// SIMATIC S7-200 project (STEP 7-Micro/WIN), CPU 224 REL 01.12

ORGANIZATION_BLOCK 主程序:OB1
TITLE=项目详解
// 系统通过启动按钮启动运行，首先打开进料阀门让棉条进入处理槽，进料过程中由液位传感器实时监控液位，确保液位不超过预设值以防止溢出。进料启用标志只有在液位传感器未检测到满液位且液位未满标志未置位时才会置位。进料完成后，搅拌电机在进料阀门关闭且温度适宜时启动，进行棉条的均匀分布，搅拌时间由搅拌延时定时器精确控制。细纱机运行状态在系统启动后保持置位，直到急停或故障发生。
// 在拉伸纺纱阶段，罗拉电机启动负责拉伸棉条。罗拉电机启动或罗拉电机停止前，纱架升起必须已经置位，以确保棉条正确引导至罗拉，避免纱线断裂。纱架升起在温度传感器1和定时器条件下置位，纱架降下在温度传感器2和定时器条件下置位。若特定标志位置位且定时器未超时，冷却器激活；加热器在进料阀门关闭且温度适宜时启动。出料阀门在标志位复位后开启，以输出纺好的细纱。
BEGIN
Network 1 // 网络标题
// 网络注释
LD     I0.4
O      Q0.0
=      M30.0
?000
Network 2
LD     SM0.1
MOVW   +5001, VW4000
Network 3
LD     M30.0
AN     T102
A      I0.3
=      Q0.0
Network 4
LD     M30.0
LD     I0.4
O      Q0.1
ALD
A      I1.1
AN     Q0.2
A      I0.3
=      Q0.1
Network 5
LD     M30.0
AN     I1.1
AN     M0.0
=      M30.1
Network 6
LD     M30.1
LD     I0.5
O      Q1.0
ALD
=      M30.2
Network 7
LD     M30.2
AN     Q1.1
AN     C1
AN     I0.6
=      Q1.0
Network 8
LD     M30.1
LD     I0.6
O      C1
O      Q1.1
ALD
AN     Q1.0
=      Q1.1
Network 9
LD     Q0.0
LD     I0.7
O      M0.2
ALD
=      M0.2
Network 10
LD     Q0.0
LD     I1.0
O      I1.2
O      M0.2
O      M0.3
O      M6.6
O      M6.7
ALD
=      M0.3
Network 11
LD     Q0.0
LD     I1.5
O      M0.0
ALD
LD     M0.2
O      M0.3
ALD
=      M0.0
Network 12
LD     Q0.0
LD     I1.5
O      M0.0
ALD
LD     M0.2
O      M0.3
ALD
AW=    VW1058, +2
TON    T108, VW1018
TON    T109, VW1020
Network 13
LD     Q0.0
LD     I2.0
AW=    VW1058, +1
LD     T108
AW=    VW1058, +2
OLD
O      Q0.2
ALD
AN     M0.2
AN     Q0.1
A      I1.3
A      M0.3
=      Q0.2
Network 14
LD     Q0.0
LD     I2.1
A      M0.3
AW=    VW1058, +1
LD     T109
A      M0.3
AW=    VW1058, +2
OLD
O      Q0.6
ALD
A      M0.0
=      Q0.6
Network 15
LD     Q0.0
LD     I2.1
A      M0.3
O      Q0.6
ALD
TON    T102, +200
Network 16
LD     Q0.0
A      M0.3
AN     T103
=      Q2.1
Network 17
LD     Q0.0
A      Q1.0
=      Q2.3
Network 18
LD     Q0.0
A      Q1.1
=      Q2.2
Network 19
LD     Q0.0
A      M0.3
AN     T104
TON    T103, +20
Network 20
LD     Q0.0
A      T103
TON    T104, +20
Network 21
LD     Q1.1
O      Q1.0
A      Q0.0
AN     M0.3
=      Q0.3
Network 22
LD     T105
EU
O      M0.5
A      Q0.0
=      M0.5
Network 23
LD     Q0.0
A      I2.2
LD     I2.3
O      Q0.4
O      Q1.1
ALD
AN     M0.3
=      Q0.4
Network 24
LD     M0.3
AN     M0.2
O      I2.5
O      Q0.7
AN     Q0.1
A      I2.6
=      Q0.5
=      Q0.7
Network 25
LD     SM0.1
BMW    VW800, VW1000, 65
R      M10.0, 8
R      M26.0, 1
R      M11.0, 2
MOVD   +0, VD20
MOVW   +0, VW24
Network 26
LD     SM0.1
O      M26.0
MOVD   +0, VD20
MOVW   +0, VW24
MOVB   8, VB20
MOVD   VD1036, VD123
R      M26.0, 1
Network 27
LD     M10.0
AN     M11.0
AN     M11.1
AN     V24.4
MOVD   +0, VD20
MOVW   +0, VW24
MOVB   16#80, VB20
MOVD   VD1040, VD43
R      M10.0, 8
Network 28
LD     M10.1
AN     M11.0
AN     M11.1
AN     V24.4
MOVD   +0, VD20
MOVW   +0, VW24
MOVB   16#40, VB20
MOVD   VD1044, VD63
R      M10.0, 8
Network 29
LD     M10.2
AN     M11.0
AN     M11.1
AN     V24.4
MOVD   +0, VD20
MOVW   +0, VW24
MOVB   16#20, VB20
MOVD   VD1048, VD83
R      M10.0, 8
Network 30
LD     M10.3
AN     M11.0
AN     M11.1
AN     V24.4
MOVD   +0, VD20
MOVW   +0, VW24
MOVB   16#10, VB20
MOVD   VD1052, VD103
R      M10.0, 8
Network 31
LD     M10.4
AN     M11.0
AN     M11.1
AN     V24.4
MOVD   +0, VD20
MOVW   +0, VW24
MOVB   8, VB20
MOVD   VD1036, VD123
R      M10.0, 8
Network 32
LD     M10.5
AN     M11.0
AN     M11.1
AN     V24.4
MOVD   +0, VD20
MOVW   +0, VW24
MOVB   4, VB20
MOVW   VW1000, VW147
R      M10.0, 8
Network 33
LD     V145.2
AW<=   VW147, +4
AW>=   VW147, +1
MOVW   VW147, VW1000
MOVW   VW147, VW800
MOVW   +800, SMW32
MOVB   16#82, SMB31
MOVW   16#1, MW9
MOVW   VW1000, AC0
DECW   AC0
SLW    MW9, AC0
R      V145.2, 1
Network 34
LD     V145.2
LDW>=  VW147, +5
OW=    VW147, +0
ALD
MOVB   8, VB24
R      V145.2, 1
Network 35
LD     M10.6
EU
S      M11.0, 1
Network 36
LDN    V20.0
AB=    VB21, 0
=      M26.2
Network 37
LD     M10.6
AN     M11.1
AN     V24.4
A      M26.2
MOVD   +0, VD20
MOVW   +0, VW24
MOVB   2, VB20
R      M10.0, 8
Network 38
LD     V168.1
MOVW   VW1030, VW182
MOVB   1, VB20
R      V168.1, 1
Network 39
LD     V180.1
MOVW   VW1022, VW202
MOVB   16#80, VB21
R      V180.1, 1
Network 40
LD     V200.1
MOVW   VW1024, VW222
MOVB   16#40, VB21
R      V200.1, 1
Network 41
LD     V220.1
MOVW   VW1026, VW244
MOVB   16#20, VB21
R      V220.1, 1
Network 42
LD     V242.1
MOVW   VW1056, VW263
MOVB   16#10, VB21
R      V242.1, 1
Network 43
LD     V261.1
MOVW   VW1032, VW284
MOVB   8, VB21
R      V261.1, 1
Network 44
LD     V282.1
MOVW   VW1034, VW300
MOVB   4, VB21
R      V282.1, 1
Network 45
LD     V298.1
MOVD   VD5000, VD324
MOVB   2, VB21
R      V298.1, 1
Network 46
LD     V322.1
MOVB   1, VB21
R      V322.1, 1
Network 47
LD     V346.1
S      M26.0, 1
R      M11.0, 1
R      V346.1, 1
R      M10.0, 8
Network 48
LD     I2.4
EU
R      V723.2, 1
R      V402.2, 1
R      V422.2, 1
R      V442.2, 1
R      V462.2, 1
R      V482.2, 1
R      V502.2, 1
R      V522.2, 1
R      V543.2, 1
R      V561.2, 1
R      V580.2, 1
R      V602.2, 1
R      V622.2, 1
R      V642.2, 1
R      V663.2, 1
R      V686.2, 1
R      V703.2, 1
Network 49
LDB>=  VB22, 1
AB<=   VB22, 16#40
OB>=   VB23, 1
OB>=   VB24, 16#10
AN     I2.4
MOVB   4, VB24
Network 50
LDN    I2.4
AN     M11.1
MOVW   +0, VW22
R      V24.4, 4
Network 51
LDN    I2.4
AB=    VB22, 16#80
MOVB   4, VB24
R      V22.7, 1
Network 52
LDN    I2.4
AB=    VB22, 16#40
MOVB   4, VB24
R      V22.6, 1
R      M11.1, 1
Network 53
LD     M10.7
AN     I2.4
MOVD   +0, VD20
MOVW   +0, VW24
MOVB   4, VB24
R      M10.0, 8
Network 54
LD     M10.7
A      I2.4
AN     M11.0
AN     V24.4
MOVD   +0, VD20
MOVW   +0, VW24
MOVB   16#80, VB22
R      M10.0, 8
S      M11.1, 1
Network 55
LD     V368.1
A      I2.4
MOVB   16#40, VB22
R      V368.1, 1
Network 56
LD     V368.1
AN     I2.4
R      V368.1, 1
R      M11.1, 1
R      M10.0, 8
Network 57
LD     V386.2
A      M11.1
A      I2.4
AW<=   VW388, +17
AW>=   VW388, +1
MOVD   +0, VD22
MOVB   16#20, VB22
DECW   VW388
SRD    VD22, VB389
MOVW   +0, VW388
R      V386.2, 1
R      M11.1, 1
R      M10.0, 8
Network 58
LD     V386.2
A      I2.4
LDW>=  VW388, +18
OW=    VW388, +0
ALD
MOVB   8, VB24
MOVW   +0, VW388
R      V386.2, 1
R      M11.1, 1
R      M10.0, 8
Network 59
LD     V386.2
AN     I2.4
R      V386.2, 1
R      M11.1, 1
R      M10.0, 8
Network 60
LDB>=  VB22, 1
AB<=   VB22, 16#20
OB>=   VB23, 1
OB>=   VB24, 16#20
EU
MOVD   VD1040, VD404
MOVD   VD1044, VD424
MOVD   VD1048, VD444
MOVD   VD1052, VD464
MOVD   VD1036, VD484
MOVW   VW1002, VW504
MOVW   VW1004, VW524
MOVW   VW1028, VW545
Network 61
LDB>=  VB22, 1
AB<=   VB22, 16#20
OB>=   VB23, 1
OB>=   VB24, 16#20
EU
MOVD   VD1006, VD563
MOVW   VW1056, VW582
MOVW   VW1014, VW604
MOVW   VW1016, VW624
MOVW   VW1012, VW644
MOVW   VW1010, VW665
MOVW   VW1058, VW688
MOVW   VW1018, VW705
MOVW   VW1020, VW725
Network 62
LD     V402.2
A      I2.4
AD=    VD404, +0
MOVD   VD404, VD1040
MOVD   VD404, VD840
MOVW   +840, SMW32
MOVB   16#83, SMB31
MOVB   16#10, VB22
R      V402.2, 1
Network 63
LD     V402.2
A      I2.4
AD>=   VD404, +1
MOVB   8, VB24
R      V402.2, 1
Network 64
LD     V422.2
A      I2.4
AD=    VD424, +0
MOVD   VD424, VD1044
MOVD   VD424, VD844
MOVW   +844, SMW32
MOVB   16#83, SMB31
MOVB   8, VB22
R      V422.2, 1
Network 65
LD     V422.2
A      I2.4
AD>=   VD424, +1
MOVB   8, VB24
R      V422.2, 1
Network 66
LD     V442.2
A      I2.4
AD=    VD444, +0
MOVD   VD444, VD1048
MOVD   VD444, VD848
MOVW   +848, SMW32
MOVB   16#83, SMB31
MOVB   4, VB22
R      V442.2, 1
Network 67
LD     V442.2
A      I2.4
AD>=   VD444, +1
MOVB   8, VB24
R      V442.2, 1
Network 68
LD     V462.2
A      I2.4
AD=    VD464, +0
MOVD   VD464, VD1052
MOVD   VD464, VD852
MOVW   +852, SMW32
MOVB   16#83, SMB31
MOVB   2, VB22
R      V462.2, 1
Network 69
LD     V462.2
A      I2.4
AD>=   VD464, +1
MOVB   8, VB24
R      V462.2, 1
Network 70
LD     V482.2
A      I2.4
AD=    VD484, +0
MOVD   VD484, VD1036
MOVD   VD484, VD836
MOVW   +836, SMW32
MOVB   16#83, SMB31
MOVB   1, VB22
R      V482.2, 1
Network 71
LD     V482.2
A      I2.4
AD>=   VD484, +1
MOVB   8, VB24
R      V482.2, 1
Network 72
LD     V502.2
A      I2.4
LDW=   VW504, +205
OW=    VW504, +220
OW=    VW504, +240
ALD
MOVW   VW504, VW1002
MOVW   VW504, VW802
MOVW   +802, SMW32
MOVB   16#82, SMB31
MOVB   16#80, VB23
R      V502.2, 1
Network 73
LD     V502.2
A      I2.4
LDW>=  VW504, +206
OW<=   VW504, +219
OW>=   VW504, +221
OW<=   VW504, +239
OW>=   VW504, +241
OW<=   VW504, +204
ALD
MOVB   8, VB24
R      V502.2, 1
Network 74
LD     V522.2
A      I2.4
LDW=   VW524, +200
OW=    VW524, +250
ALD
MOVW   VW524, VW1004
MOVW   VW524, VW804
MOVW   +804, SMW32
MOVB   16#82, SMB31
MOVB   16#40, VB23
R      V522.2, 1
Network 75
LD     V522.2
A      I2.4
LDW>=  VW524, +201
OW<=   VW524, +249
OW>=   VW524, +251
OW<=   VW524, +199
ALD
MOVB   8, VB24
R      V522.2, 1
Network 76
LD     V543.2
A      I2.4
LDW=   VW545, +25
OW=    VW545, +27
ALD
MOVW   VW545, VW1028
MOVW   VW545, VW828
MOVW   +828, SMW32
MOVB   16#82, SMB31
MOVB   16#20, VB23
R      V543.2, 1
Network 77
LD     V543.2
A      I2.4
LDW>=  VW545, +28
OW<=   VW545, +24
ALD
MOVB   8, VB24
R      V543.2, 1
Network 78
LD     V561.2
A      I2.4
AD<=   VD563, +99999
MOVD   VD563, VD1006
MOVD   VD563, VD806
MOVW   +806, SMW32
MOVB   16#83, SMB31
MOVB   16#10, VB23
R      V561.2, 1
Network 79
LD     V561.2
A      I2.4
AD>=   VD563, +100000
MOVB   8, VB24
R      V561.2, 1
Network 80
LD     V580.2
A      I2.4
AW<=   VW582, +999
MOVW   VW582, VW1056
MOVW   VW582, VW856
MOVW   +856, SMW32
MOVB   16#82, SMB31
MOVB   8, VB23
R      V580.2, 1
Network 81
LD     V580.2
A      I2.4
AW>=   VW582, +1000
MOVB   8, VB24
R      V580.2, 1
Network 82
LD     V602.2
A      I2.4
AW<=   VW604, +99
MOVW   VW604, VW1014
MOVW   VW604, VW814
MOVW   +814, SMW32
MOVB   16#82, SMB31
MOVB   4, VB23
R      V602.2, 1
Network 83
LD     V602.2
A      I2.4
AW>=   VW604, +100
MOVB   8, VB24
R      V602.2, 1
Network 84
LD     V622.2
A      I2.4
LDW=   VW624, +1
OW=    VW624, +2
ALD
MOVW   VW624, VW1016
MOVW   VW624, VW816
MOVW   +816, SMW32
MOVB   16#82, SMB31
MOVB   2, VB23
R      V622.2, 1
Network 85
LD     V622.2
A      I2.4
LDW>=  VW624, +3
OW<=   VW624, +0
ALD
MOVB   8, VB24
R      V622.2, 1
Network 86
LD     V642.2
A      I2.4
AW<=   VW644, +600
MOVW   VW644, VW1012
MOVW   VW644, VW812
MOVW   +812, SMW32
MOVB   16#82, SMB31
MOVB   1, VB23
R      V642.2, 1
Network 87
LD     V642.2
A      I2.4
AW>=   VW644, +601
MOVB   8, VB24
R      V642.2, 1
Network 88
LD     V663.2
A      I2.4
AW<=   VW665, +1999
MOVW   VW665, VW1010
MOVW   VW665, VW810
MOVW   +810, SMW32
MOVB   16#82, SMB31
MOVB   16#80, VB24
R      V663.2, 1
Network 89
LD     V663.2
A      I2.4
AW>=   VW665, +2000
MOVB   8, VB24
R      V663.2, 1
Network 90
LD     V686.2
A      I2.4
LDW=   VW688, +2
OW=    VW688, +1
ALD
MOVW   VW688, VW1058
MOVW   VW688, VW858
MOVW   +858, SMW32
MOVB   16#82, SMB31
MOVB   16#40, VB24
R      V686.2, 1
Network 91
LD     V686.2
A      I2.4
LDW>=  VW688, +3
OW=    VW688, +0
ALD
MOVB   8, VB24
R      V686.2, 1
Network 92
LD     V703.2
A      I2.4
AW<=   VW705, +99
MOVW   VW705, VW1018
MOVW   VW705, VW818
MOVW   +818, SMW32
MOVB   16#82, SMB31
MOVB   16#20, VB24
R      V703.2, 1
Network 93
LD     V703.2
A      I2.4
AW>=   VW705, +100
MOVB   8, VB24
R      V703.2, 1
Network 94
LD     V723.2
A      I2.4
AW<=   VW725, +999
MOVW   VW725, VW1020
MOVW   VW725, VW820
MOVW   +820, SMW32
MOVB   16#82, SMB31
MOVB   16#10, VB24
R      V723.2, 1
Network 95
LD     V723.2
A      I2.4
AW>=   VW725, +1000
MOVB   8, VB24
R      V723.2, 1
Network 96
LD     V747.1
A      I2.4
S      M26.0, 1
R      M10.0, 8
R      V747.1, 1
R      V24.4, 1
Network 97
LD     V24.3
O      V24.2
AB=    MB10, 0
TON    T37, +30
Network 98
LD     T37
S      M26.0, 1
Network 99
LD     Q1.0
O      Q1.1
AN     M6.0
TON    T110, +600
Network 100
LD     T110
EU
=      M6.0
Network 101
LD     Q1.0
O      Q1.1
AN     M2.0
TON    T125, +60
Network 102
LD     T125
EU
=      M2.0
Network 103
LD     Q1.0
O      Q1.1
AN     M2.4
TON    T126, +6
Network 104
LD     T126
EU
=      M2.4
Network 105
LD     Q1.0
O      Q1.1
EU
=      M6.1
Network 106
LD     Q1.0
O      Q1.1
A      I0.1
EU
INCW   VW2000
INCW   VW2018
Network 107
LD     Q1.0
O      Q1.1
A      I0.2
EU
INCW   VW2004
Network 108
LDW>=  VW2004, +10
MOVW   VW2000, VW2008
MOVW   VW2000, VW2030
MOVW   +0, VW2004
MOVW   +10, VW2010
MUL    VW2008, VD2008
MOVW   VW2010, VW1024
MOVW   VW1024, VW222
MOVW   +0, VW2000
=      M6.2
Network 109
LD     M6.1
MOVW   +0, VW2008
MOVW   +0, VW2030
MOVW   +0, VW2004
MOVW   +0, VW2012
MOVW   +0, VW2000
Network 110
LD     M6.0
MOVW   VW1004, VW2202
DIV    +10, VD2200
Network 111
LD     M6.0
MUL    VW1010, VD2200
MOVW   VW1002, VW2402
MUL    +2, VD2400
DIV    +10, VD2400
DIV    VW2402, VD2200
MUL    VW2012, VD2200
SRD    VD2200, 6
DIV    +10, VD2200
MOVD   VD2200, VD2404
MUL    +13, VD2404
DIV    +5, VD2200
-I     VW2202, VW2406
MOVW   +0, VW2012
MOVW   VW2406, VW1030
MOVW   VW1030, VW182
MOVW   VW1030, VW830
Network 112
LD     M6.0
MOVW   VW2018, VW1022
MOVW   VW1022, VW202
MOVW   VW1022, VW822
MOVW   +0, VW2018
Network 113
LD     M6.0
MOVW   VW1030, VW2216
DIV    VW1022, VD2214
MUL    +129, VD2214
MOVW   VW2216, VW1032
MOVW   VW1032, VW284
MOVW   VW1032, VW832
Network 114
LD     M6.2
MOVW   VW1056, VW2206
MUL    +10, VD2204
Network 115
LD     M6.2
DIV    VW2030, VD2204
MOVW   VW2030, VW2504
MOVW   VW2204, VW2502
MUL    +100, VD2500
MUL    +100, VD2204
MOVW   VW2206, VW1026
MOVW   VW1026, VW244
MOVW   VW1026, VW826
Network 116
LD     M6.2
AW>=   VW2504, +256
SRW    VW2504, 1
SRD    VD2500, 1
Network 117
LD     M6.2
DIV    VW2504, VD2500
+I     VW2502, VW1026
MOVW   VW1026, VW244
MOVW   VW1026, VW826
Network 118
LD     M6.0
MOVW   +472, VW2212
MUL    VW1022, VD2210
SRD    VD2210, 3
DIV    +25, VD2210
MUL    VW1026, VD2210
SRD    VD2210, 6
DIV    +25, VD2210
SLD    VD2210, 5
MOVW   VW2212, VW1034
MOVW   VW1034, VW300
MOVW   VW1034, VW834
Network 119
LD     I0.1
EU
INCW   VW2034
Network 120
LDW>=  VW2034, +10
=      M6.3
MOVW   +0, VW2034
Network 121
LD     M6.3
AW=    VW545, +25
+I     +785, VW2300
Network 122
LD     M6.3
AW=    VW545, +27
+I     +846, VW2300
Network 123
LD     M6.3
AW=    VW624, +1
AW>=   VW2300, +1000
-I     +1000, VW2300
INCD   VD2310
MOVD   VD2310, VD324
=      M6.4
Network 124
LD     M6.3
AW=    VW545, +25
+D     +785, VD1036
MOVD   VD1036, VD123
MOVD   VD1036, VD836
Network 125
LD     M6.3
AW=    VW545, +27
+D     +846, VD1036
MOVD   VD1036, VD123
MOVD   VD1036, VD836
Network 126
LDW=   VW624, +1
AD>=   VD2310, VD1006
=      M6.6
Network 127
LD     M6.0
EU
AW=    VW624, +2
INCW   VW2680
MOVD   VD2678, VD324
=      M2.1
Network 128
LD     M2.1
AW>=   VW2680, VW644
AW=    VW624, +2
=      M6.7
MOVW   +0, VW2680
MOVW   +0, VW2686
Network 129
LDW=   VW624, +1
MOVD   VD2310, VD5000
Network 130
LDW=   VW624, +2
MOVD   VD2678, VD5000
Network 131
LD     M2.0
EU
AW=    VW624, +2
INCW   VW2686
Network 132
LD     Q0.2
EU
MOVW   +0, VW2300
MOVD   +0, VD2310
MOVD   +0, VD2678
MOVW   +0, VW2686
Network 133
LD     M6.3
AD>=   VD1036, +99999000
MOVD   +0, VD1036
Network 134
LD     M6.3
AB=    VB1001, 1
AW=    VW545, +25
+D     +785, VD1040
=      M8.0
Network 135
LD     M6.3
AB=    VB1001, 1
AW=    VW545, +27
+D     +846, VD1040
=      M8.1
Network 136
LD     M8.0
O      M8.1
MOVD   VD1040, VD43
MOVD   VD1040, VD840
=      M8.2
Network 137
LD     M8.2
AD>=   VD1040, +99999000
MOVD   +0, VD1040
Network 138
LD     M6.3
AB=    VB1001, 2
AW=    VW545, +25
+D     +785, VD1044
=      M8.3
Network 139
LD     M6.3
AB=    VB1001, 2
AW=    VW545, +27
+D     +846, VD1044
=      M8.4
Network 140
LD     M8.3
O      M8.4
MOVD   VD1044, VD63
MOVD   VD1044, VD844
=      M8.5
Network 141
LD     M8.5
AD>=   VD1044, +99999000
MOVD   +0, VD1044
Network 142
LD     M6.3
AB=    VB1001, 3
AW=    VW545, +25
+D     +785, VD1048
=      M8.6
Network 143
LD     M6.3
AB=    VB1001, 3
AW=    VW545, +27
+D     +846, VD1048
=      M8.7
Network 144
LD     M8.6
O      M8.7
MOVD   VD1048, VD83
MOVD   VD1048, VD848
=      M9.0
Network 145
LD     M9.0
AD>=   VD1048, +99999000
MOVD   +0, VD1048
Network 146
LD     M6.3
AB=    VB1001, 4
AW=    VW545, +25
+D     +785, VD1052
=      M9.1
Network 147
LD     M6.3
AB=    VB1001, 4
AW=    VW545, +27
+D     +846, VD1052
=      M9.2
Network 148
LD     M9.1
O      M9.2
MOVD   VD1052, VD103
MOVD   VD1052, VD852
=      M9.4
Network 149
LD     M9.4
AD>=   VD1052, +99999000
MOVD   +0, VD1052
Network 150
LD     Q1.0
A      M6.0
A      I2.7
LD     Q1.1
CTU    C1, VW1014
Network 151
LD     SM0.1
ATCH   INT1:INT1, 0
ENI
END_ORGANIZATION_BLOCK

INTERRUPT_BLOCK INT1:INT1
TITLE=
BEGIN
Network 2
LD     SM0.0
INCW   VW2012
END_INTERRUPT_BLOCK

DATA_BLOCK_TAB 用户定义1
BEGIN
VB0      16#54
VB1      16#44
VB2      16#60
VB3      16#40
VB4      16#26
VB5      16#A
VB6      16#0
VB7      16#1E
VB8      16#0
VB9      16#14
VB10     16#7
VB11     16#D0
VB12     16#1
VB13     16#0
VB14     16#0
VB15     16#0
VB16     16#0
VB17     16#0
VB18     16#0
VB19     16#0
VB20     16#0
VB21     16#0
VB22     16#0
VB23     16#0
VB24     16#0
VB25     16#0
VB26     16#0
VB27     16#0
VB28     16#0
VB29     16#0
VB30     16#41
VB31     16#20
VB32     16#B0
VB33     16#E0
VB34     16#B0
VB35     16#E0
VB36     16#B2
VB37     16#FA
VB38     16#20
VB39     16#20
VB40     16#20
VB41     16#0
VB42     16#23
VB43     16#0
VB44     16#0
VB45     16#0
VB46     16#0
VB47     16#20
VB48     16#6D
VB49     16#20
VB50     16#42
VB51     16#20
VB52     16#B0
VB53     16#E0
VB54     16#B0
VB55     16#E0
VB56     16#B2
VB57     16#FA
VB58     16#20
VB59     16#20
VB60     16#20
VB61     16#0
VB62     16#23
VB63     16#0
VB64     16#0
VB65     16#0
VB66     16#0
VB67     16#20
VB68     16#6D
VB69     16#20
VB70     16#43
VB71     16#20
VB72     16#B0
VB73     16#E0
VB74     16#B0
VB75     16#E0
VB76     16#B2
VB77     16#FA
VB78     16#20
VB79     16#20
VB80     16#20
VB81     16#0
VB82     16#23
VB83     16#0
VB84     16#0
VB85     16#0
VB86     16#0
VB87     16#20
VB88     16#6D
VB89     16#20
VB90     16#44
VB91     16#20
VB92     16#B0
VB93     16#E0
VB94     16#B0
VB95     16#E0
VB96     16#B2
VB97     16#FA
VB98     16#20
VB99     16#20
VB100    16#20
VB101    16#0
VB102    16#23
VB103    16#0
VB104    16#0
VB105    16#0
VB106    16#0
VB107    16#20
VB108    16#6D
VB109    16#20
VB110    16#D7
VB111    16#DC
VB112    16#B3
VB113    16#A4
VB114    16#20
VB115    16#20
VB116    16#20
VB117    16#20
VB118    16#20
VB119    16#20
VB120    16#20
VB121    16#0
VB122    16#23
VB123    16#0
VB124    16#0
VB125    16#0
VB126    16#0
VB127    16#20
VB128    16#6D
VB129    16#20
VB130    16#B5
VB131    16#B1
VB132    16#C7
VB133    16#B0
VB134    16#B0
VB135    16#E0
VB136    16#C9
VB137    16#E8
VB138    16#B6
VB139    16#A8
VB140    16#20
VB141    16#20
VB142    16#20
VB143    16#20
VB144    16#20
VB145    16#10
VB146    16#10
VB147    16#0
VB148    16#1
VB149    16#20
VB150    16#20
VB151    16#20
VB152    16#20
VB153    16#20
VB154    16#20
VB155    16#20
VB156    16#CF
VB157    16#D4
VB158    16#CA
VB159    16#BE
VB160    16#B2
VB161    16#CE
VB162    16#CA
VB163    16#FD
VB164    16#20
VB165    16#20
VB166    16#20
VB167    16#20
VB168    16#1
VB169    16#0
VB170    16#31
VB171    16#2E
VB172    16#B6
VB173    16#A7
VB174    16#CB
VB175    16#D9
VB176    16#20
VB177    16#20
VB178    16#20
VB179    16#20
VB180    16#1
VB181    16#10
VB182    16#0
VB183    16#0
VB184    16#20
VB185    16#72
VB186    16#2F
VB187    16#6D
VB188    16#69
VB189    16#6E
VB190    16#32
VB191    16#2E
VB192    16#C2
VB193    16#DE
VB194    16#C0
VB195    16#AD
VB196    16#CB
VB197    16#D9
VB198    16#B6
VB199    16#C8
VB200    16#1
VB201    16#10
VB202    16#0
VB203    16#0
VB204    16#20
VB205    16#72
VB206    16#2F
VB207    16#6D
VB208    16#69
VB209    16#6E
VB210    16#33
VB211    16#C7
VB212    16#A3
VB213    16#C9
VB214    16#EC
VB215    16#B1
VB216    16#B6
VB217    16#CA
VB218    16#FD
VB219    16#20
VB220    16#1
VB221    16#12
VB222    16#0
VB223    16#0
VB224    16#20
VB225    16#B1
VB226    16#B6
VB227    16#20
VB228    16#20
VB229    16#20
VB230    16#34
VB231    16#2E
VB232    16#CF
VB233    16#B8
VB234    16#C9
VB235    16#B4
VB236    16#BA
VB237    16#C5
VB238    16#CA
VB239    16#FD
VB240    16#20
VB241    16#20
VB242    16#1
VB243    16#12
VB244    16#0
VB245    16#0
VB246    16#67
VB247    16#2F
VB248    16#6B
VB249    16#6D
VB250    16#35
VB251    16#2E
VB252    16#B4
VB253    16#D6
VB254    16#C9
VB255    16#B4
VB256    16#B6
VB257    16#A8
VB258    16#C1
VB259    16#BF
VB260    16#20
VB261    16#1
VB262    16#10
VB263    16#0
VB264    16#0
VB265    16#20
VB266    16#67
VB267    16#2F
VB268    16#6B
VB269    16#6D
VB270    16#36
VB271    16#2E
VB272    16#C4
VB273    16#ED
VB274    16#B6
VB275    16#C8
VB276    16#20
VB277    16#20
VB278    16#20
VB279    16#20
VB280    16#20
VB281    16#20
VB282    16#1
VB283    16#11
VB284    16#0
VB285    16#0
VB286    16#20
VB287    16#74
VB288    16#2F
VB289    16#6D
VB290    16#37
VB291    16#2E
VB292    16#50
VB293    16#2D
VB294    16#2D
VB295    16#20
VB296    16#20
VB297    16#20
VB298    16#1
VB299    16#13
VB300    16#0
VB301    16#0
VB302    16#20
VB303    16#6B
VB304    16#67
VB305    16#2F
VB306    16#6B
VB307    16#73
VB308    16#2E
VB309    16#68
VB310    16#38
VB311    16#2E
VB312    16#BC
VB313    16#C6
VB314    16#B3
VB315    16#A4
VB316    16#20
VB317    16#20
VB318    16#20
VB319    16#20
VB320    16#20
VB321    16#20
VB322    16#1
VB323    16#20
VB324    16#0
VB325    16#0
VB326    16#0
VB327    16#0
VB328    16#20
VB329    16#6D
VB330    16#20
VB331    16#20
VB332    16#20
VB333    16#20
VB334    16#20
VB335    16#CF
VB336    16#D4
VB337    16#CA
VB338    16#BE
VB339    16#BD
VB340    16#E1
VB341    16#CA
VB342    16#F8
VB343    16#20
VB344    16#20
VB345    16#20
VB346    16#1
VB347    16#0
VB348    16#0
VB349    16#0
VB350    16#20
VB351    16#20
VB352    16#20
VB353    16#20
VB354    16#20
VB355    16#C9
VB356    16#E8
VB357    16#D6
VB358    16#C3
VB359    16#B2
VB360    16#CE
VB361    16#CA
VB362    16#FD
VB363    16#20
VB364    16#20
VB365    16#20
VB366    16#20
VB367    16#20
VB368    16#1
VB369    16#0
VB370    16#CA
VB371    16#E4
VB372    16#C8
VB373    16#EB
VB374    16#B2
VB375    16#CE
VB376    16#CA
VB377    16#FD
VB378    16#B4
VB379    16#FA
VB380    16#C2
VB381    16#EB
VB382    16#20
VB383    16#20
VB384    16#20
VB385    16#20
VB386    16#10
VB387    16#10
VB388    16#0
VB389    16#0
VB390    16#31
VB391    16#2E
VB392    16#41
VB393    16#20
VB394    16#B0
VB395    16#E0
VB396    16#20
VB397    16#20
VB398    16#20
VB399    16#20
VB400    16#20
VB401    16#20
VB402    16#10
VB403    16#23
VB404    16#0
VB405    16#0
VB406    16#0
VB407    16#0
VB408    16#20
VB409    16#6D
VB410    16#32
VB411    16#2E
VB412    16#42
VB413    16#20
VB414    16#B0
VB415    16#E0
VB416    16#20
VB417    16#20
VB418    16#20
VB419    16#20
VB420    16#20
VB421    16#20
VB422    16#10
VB423    16#23
VB424    16#0
VB425    16#0
VB426    16#0
VB427    16#0
VB428    16#20
VB429    16#6D
VB430    16#33
VB431    16#2E
VB432    16#43
VB433    16#20
VB434    16#B0
VB435    16#E0
VB436    16#20
VB437    16#20
VB438    16#20
VB439    16#20
VB440    16#20
VB441    16#20
VB442    16#10
VB443    16#23
VB444    16#0
VB445    16#0
VB446    16#0
VB447    16#0
VB448    16#20
VB449    16#6D
VB450    16#34
VB451    16#2E
VB452    16#44
VB453    16#20
VB454    16#B0
VB455    16#E0
VB456    16#20
VB457    16#20
VB458    16#20
VB459    16#20
VB460    16#20
VB461    16#20
VB462    16#10
VB463    16#23
VB464    16#0
VB465    16#0
VB466    16#0
VB467    16#0
VB468    16#20
VB469    16#6D
VB470    16#35
VB471    16#2E
VB472    16#D7
VB473    16#DC
VB474    16#B3
VB475    16#A4
VB476    16#20
VB477    16#20
VB478    16#20
VB479    16#20
VB480    16#20
VB481    16#20
VB482    16#10
VB483    16#23
VB484    16#0
VB485    16#0
VB486    16#0
VB487    16#0
VB488    16#20
VB489    16#6D
VB490    16#36
VB491    16#2E
VB492    16#B6
VB493    16#A7
VB494    16#C5
VB495    16#CC
VB496    16#D6
VB497    16#B1
VB498    16#BE
VB499    16#B6
VB500    16#20
VB501    16#20
VB502    16#10
VB503    16#11
VB504    16#0
VB505    16#0
VB506    16#20
VB507    16#20
VB508    16#6D
VB509    16#6D
VB510    16#37
VB511    16#2E
VB512    16#B9
VB513    16#F6
VB514    16#C5
VB515    16#CC
VB516    16#D6
VB517    16#B1
VB518    16#BE
VB519    16#B6
VB520    16#20
VB521    16#20
VB522    16#10
VB523    16#10
VB524    16#0
VB525    16#0
VB526    16#20
VB527    16#20
VB528    16#6D
VB529    16#20
VB530    16#38
VB531    16#2E
VB532    16#C7
VB533    16#B0
VB534    16#C2
VB535    16#DE
VB536    16#C0
VB537    16#AD
VB538    16#D6
VB539    16#B1
VB540    16#BE
VB541    16#B6
VB542    16#20
VB543    16#10
VB544    16#10
VB545    16#0
VB546    16#0
VB547    16#20
VB548    16#6D
VB549    16#6D
VB550    16#39
VB551    16#2E
VB552    16#B6
VB553    16#A8
VB554    16#B3
VB555    16#A4
VB556    16#C9
VB557    16#E8
VB558    16#B6
VB559    16#A8
VB560    16#20
VB561    16#10
VB562    16#20
VB563    16#0
VB564    16#0
VB565    16#0
VB566    16#0
VB567    16#20
VB568    16#20
VB569    16#6D
VB570    16#31
VB571    16#30
VB572    16#B4
VB573    16#D6
VB574    16#C9
VB575    16#B4
VB576    16#B6
VB577    16#A8
VB578    16#C1
VB579    16#BF
VB580    16#10
VB581    16#10
VB582    16#0
VB583    16#0
VB584    16#20
VB585    16#67
VB586    16#2F
VB587    16#6B
VB588    16#6D
VB589    16#20
VB590    16#31
VB591    16#31
VB592    16#2E
VB593    16#C9
VB594    16#FD
VB595    16#CB
VB596    16#D9
VB597    16#CA
VB598    16#B1
VB599    16#BC
VB600    16#E4
VB601    16#20
VB602    16#10
VB603    16#10
VB604    16#0
VB605    16#0
VB606    16#20
VB607    16#6D
VB608    16#69
VB609    16#6E
VB610    16#31
VB611    16#32
VB612    16#2E
VB613    16#C4
VB614    16#A3
VB615    16#CA
VB616    16#BD
VB617    16#D1
VB618    16#A1
VB619    16#D4
VB620    16#F1
VB621    16#20
VB622    16#10
VB623    16#10
VB624    16#0
VB625    16#0
VB626    16#20
VB627    16#20
VB628    16#20
VB629    16#20
VB630    16#31
VB631    16#33
VB632    16#2E
VB633    16#B6
VB634    16#A8
VB635    16#CA
VB636    16#B1
VB637    16#C9
VB638    16#E8
VB639    16#B6
VB640    16#A8
VB641    16#20
VB642    16#10
VB643    16#10
VB644    16#0
VB645    16#0
VB646    16#20
VB647    16#6D
VB648    16#69
VB649    16#6E
VB650    16#31
VB651    16#34
VB652    16#2E
VB653    16#D0
VB654    16#DE
VB655    16#D5
VB656    16#FD
VB657    16#CF
VB658    16#B5
VB659    16#CA
VB660    16#FD
VB661    16#20
VB662    16#20
VB663    16#10
VB664    16#13
VB665    16#0
VB666    16#0
VB667    16#20
VB668    16#20
VB669    16#20
VB670    16#31
VB671    16#35
VB672    16#2E
VB673    16#C8
VB674    16#FD
VB675    16#D7
VB676    16#D4
VB677    16#B6
VB678    16#AF
VB679    16#D1
VB680    16#A1
VB681    16#D4
VB682    16#F1
VB683    16#20
VB684    16#20
VB685    16#20
VB686    16#10
VB687    16#10
VB688    16#0
VB689    16#0
VB690    16#31
VB691    16#36
VB692    16#2E
VB693    16#CF
VB694    16#C2
VB695    16#BD
VB696    16#B5
VB697    16#CA
VB698    16#B1
VB699    16#BC
VB700    16#E4
VB701    16#20
VB702    16#20
VB703    16#10
VB704    16#11
VB705    16#0
VB706    16#0
VB707    16#20
VB708    16#20
VB709    16#73
VB710    16#31
VB711    16#37
VB712    16#2E
VB713    16#C9
VB714    16#B2
VB715    16#B3
VB716    16#B5
VB717    16#CA
VB718    16#B1
VB719    16#BC
VB720    16#E4
VB721    16#20
VB722    16#20
VB723    16#10
VB724    16#11
VB725    16#0
VB726    16#0
VB727    16#20
VB728    16#20
VB729    16#73
VB730    16#20
VB731    16#20
VB732    16#20
VB733    16#20
VB734    16#20
VB735    16#C9
VB736    16#E8
VB737    16#D6
VB738    16#C3
VB739    16#BD
VB740    16#E1
VB741    16#CA
VB742    16#F8
VB743    16#20
VB744    16#20
VB745    16#20
VB746    16#20
VB747    16#1
VB748    16#0
VB749    16#0
VB750    16#20
VB751    16#20
VB752    16#20
VB753    16#20
VB754    16#C9
VB755    16#E8
VB756    16#D6
VB757    16#C3
VB758    16#B2
VB759    16#CE
VB760    16#CA
VB761    16#FD
VB762    16#B4
VB763    16#ED
VB764    16#CE
VB765    16#F3
VB766    16#20
VB767    16#20
VB768    16#0
VB769    16#0
VB770    16#20
VB771    16#20
VB772    16#20
VB773    16#20
VB774    16#20
VB775    16#C3
VB776    16#DC
VB777    16#C2
VB778    16#EB
VB779    16#CB
VB780    16#F8
VB781    16#B9
VB782    16#D8
VB783    16#B1
VB784    16#D5
VB785    16#20
VB786    16#20
VB787    16#20
VB788    16#0
VB789    16#0
VB790    16#20
VB791    16#20
VB792    16#20
VB793    16#20
VB794    16#20
VB795    16#20
VB796    16#20
VB797    16#20
VB798    16#20
VB799    16#20
VB800    16#0
VB801    16#2
VB802    16#0
VB803    16#DC
VB804    16#0
VB805    16#FA
VB806    16#0
VB807    16#0
VB808    16#27
VB809    16#5C
VB810    16#3
VB811    16#D5
VB812    16#0
VB813    16#78
VB814    16#0
VB815    16#2
VB816    16#0
VB817    16#1
VB818    16#0
VB819    16#5
VB820    16#0
VB821    16#32
VB822    16#0
VB823    16#0
VB824    16#0
VB825    16#0
VB826    16#0
VB827    16#0
VB828    16#0
VB829    16#19
VB830    16#0
VB831    16#0
VB832    16#0
VB833    16#0
VB834    16#0
VB835    16#0
VB836    16#0
VB837    16#0
VB838    16#0
VB839    16#0
VB840    16#0
VB841    16#0
VB842    16#0
VB843    16#0
VB844    16#0
VB845    16#0
VB846    16#0
VB847    16#0
VB848    16#0
VB849    16#0
VB850    16#0
VB851    16#0
VB852    16#0
VB853    16#0
VB854    16#0
VB855    16#0
VB856    16#2
VB857    16#9F
VB858    16#0
VB859    16#1
VB860    16#0
VB861    16#0
VB862    16#0
VB863    16#0
VB864    16#0
VB865    16#0
VB866    16#0
VB867    16#0
VB868    16#20
VB869    16#20
VB870    16#20
VB871    16#20
VB872    16#20
VB873    16#20
VB874    16#20
VB875    16#20
VB876    16#20
VB877    16#20
VB878    16#20
VB879    16#20
VB880    16#20
VB881    16#20
VB882    16#20
VB883    16#20
VB884    16#20
VB885    16#20
VB886    16#20
VB887    16#20
VB888    16#20
VB889    16#20
VB890    16#20
VB891    16#20
VB892    16#20
VB893    16#20
VB894    16#20
VB895    16#20
VB896    16#20
VB897    16#20
VB898    16#20
VB899    16#20
VB900    16#20
VB901    16#20
VB902    16#20
VB903    16#20
VB904    16#20
VB905    16#20
VB906    16#20
VB907    16#20
VB908    16#20
VB909    16#20
VB910    16#20
VB911    16#20
VB912    16#20
VB913    16#20
VB914    16#20
VB915    16#20
VB916    16#20
VB917    16#20
VB918    16#20
VB919    16#20
VB920    16#20
VB921    16#20
VB922    16#20
VB923    16#20
VB924    16#20
VB925    16#20
VB926    16#20
VB927    16#20
VB928    16#20
VB929    16#20
VB930    16#0
VB931    16#0
VB932    16#0
VB933    16#0
VB934    16#0
VB935    16#0
VB936    16#0
VB937    16#0
VB938    16#0
VB939    16#0
VB940    16#0
VB941    16#0
VB942    16#0
VB943    16#0
VB944    16#0
VB945    16#0
VB946    16#0
VB947    16#0
VB948    16#0
VB949    16#0
VB950    16#0
VB951    16#0
VB952    16#0
VB953    16#0
VB954    16#0
VB955    16#0
VB956    16#0
VB957    16#0
VB958    16#0
VB959    16#0
VB960    16#0
VB961    16#0
VB962    16#0
VB963    16#0
VB964    16#0
VB965    16#0
VB966    16#0
VB967    16#0
VB968    16#0
VB969    16#0
VB970    16#0
VB971    16#0
VB972    16#0
VB973    16#0
VB974    16#0
VB975    16#0
VB976    16#0
VB977    16#0
VB978    16#0
VB979    16#0
VB980    16#0
VB981    16#0
VB982    16#0
VB983    16#0
VB984    16#0
VB985    16#0
VB986    16#0
VB987    16#0
VB988    16#0
VB989    16#0
VB990    16#0
VB991    16#0
VB992    16#0
VB993    16#0
VB994    16#0
VB995    16#0
VB996    16#0
VB997    16#0
VB998    16#0
VB999    16#0
END_DATA_BLOCK_TAB
